(* PLC project conveyor, Dassault Systèmes ControlBuild 2024x *)
(* stored: creationDateTime 2023-10-03T11:12:56-01:00 *)

(* This module simulates the behaviour of a roller table. It takes a linear speed coming from a gear motor as input. It can be associated with equipements such as rotary plate ring, traverser, ... It can be used to shift the products that are in intercation with it. *)
FUNCTION_BLOCK equipment_library.conveyor
  VAR_INPUT
    incPositionX : REAL := 0.0;
    incPositionY : REAL := 0.0;
    incPositionZ : REAL := 0.0;
  END_VAR
  VAR_INPUT
    coordCenterX : REAL := 0.0;
    coordCenterY : REAL := 0.0;
    coordCenterZ : REAL := 0.0;
    incRotationX : REAL := 0.0;
    incRotationY : REAL := 0.0;
    incRotationZ : REAL := 0.0;
  END_VAR
  VAR_INPUT
    linearSpeed : REAL := 0.0;
  END_VAR
  VAR
    status_act_prod : DINT := 0;
    m11 : REAL := 1.0;
    m12 : REAL := 0.0;
    m13 : REAL := 0.0;
    m14 : REAL := 0.0;
    m21 : REAL := 0.0;
    m22 : REAL := 1.0;
    m23 : REAL := 0.0;
    m24 : REAL := 0.0;
    m31 : REAL := 0.0;
    m32 : REAL := 0.0;
    m33 : REAL := 1.0;
    m34 : REAL := 0.0;
    m41 : REAL := 0.0;
    m42 : REAL := 0.0;
    m43 : REAL := 0.0;
    m44 : REAL := 1.0;
    incrementPositionX : REAL := 0.0;
    incrementPositionY : REAL := 0.0;
    incrementPositionZ : REAL := 0.0;
    incShiftProduct : REAL := 0.0;
    centerRotX : REAL := 0.0;
    centerRotY : REAL := 0.0;
    centerRotZ : REAL := 0.0;
    incRotY : REAL := 0.0;
    incRotZ : REAL := 0.0;
    incRotX : REAL := 0.0;
  END_VAR
  VAR
    d_locking : BOOL := false;
    v_d_locking : BOOL := false;
  END_VAR


ACTION C_source_code:
/* ----------------------------------------------------------------	*/
/* Type : Model of Operative Behaviour					*/
/* Category :  Actors and Products						*/
/* Author : Dassault Systemes						*/
/* Update date : June 2018							*/
/* ----------------------------------------------------------------	*/
/* This module simulates the behaviour of a roller table.		*/
/* It takes a linear speed coming from a gear motor as input.		*/
/* It can  be associated with equipements such as rotary plate ring,	*/
/* traverser, ...								*/
/* It can be used to shift the products that are in interaction with	*/
/* it.										*/
/* ----------------------------------------------------------------	*/


/* ----------------------------------------------------------------	*/
/* Compute the product traverse speed					*/
/* ----------------------------------------------------------------	*/
if (!d_locking)
	incShiftProduct=(linearSpeed*CLOCK_PERIOD/1000000.0);
else
	incShiftProduct=0;

/* ----------------------------------------------------------------	*/
/* Association with an traverser : take account of the traverse 	*/
/* speed of the traverser							*/
/* ----------------------------------------------------------------	*/
if (incPositionX != 0.0) moveXBy(myself, incPositionX);
if (incPositionY != 0.0) moveYBy(myself, incPositionY);
if (incPositionZ != 0.0) moveZBy(myself, incPositionZ);

/* ----------------------------------------------------------------	*/
/* Association with a rotary plate ring : take account of the 	*/
/* rotation speed of the plate						*/
/* ----------------------------------------------------------------	*/
if ((incRotationY != 0.0) || (incRotationZ != 0.0))
	rotateBy(myself, incRotationX, incRotationY, incRotationZ, coordCenterX, coordCenterY, coordCenterZ);


/* ----------------------------------------------------------------	*/
/*  Exchange of informations with products				*/
/* ----------------------------------------------------------------	*/

/* => informations coming from rotary plate ring, ...			*/
centerRotX=coordCenterX;
centerRotY=coordCenterY;
centerRotZ=coordCenterZ;
incRotX=incRotationX;
incRotY=incRotationY;
incRotZ=incRotationZ;

/* => informations coming from traverser, ...				*/
incrementPositionX=incPositionX;
incrementPositionY=incPositionY;
incrementPositionZ=incPositionZ;
END_ACTION
END_FUNCTION_BLOCK
